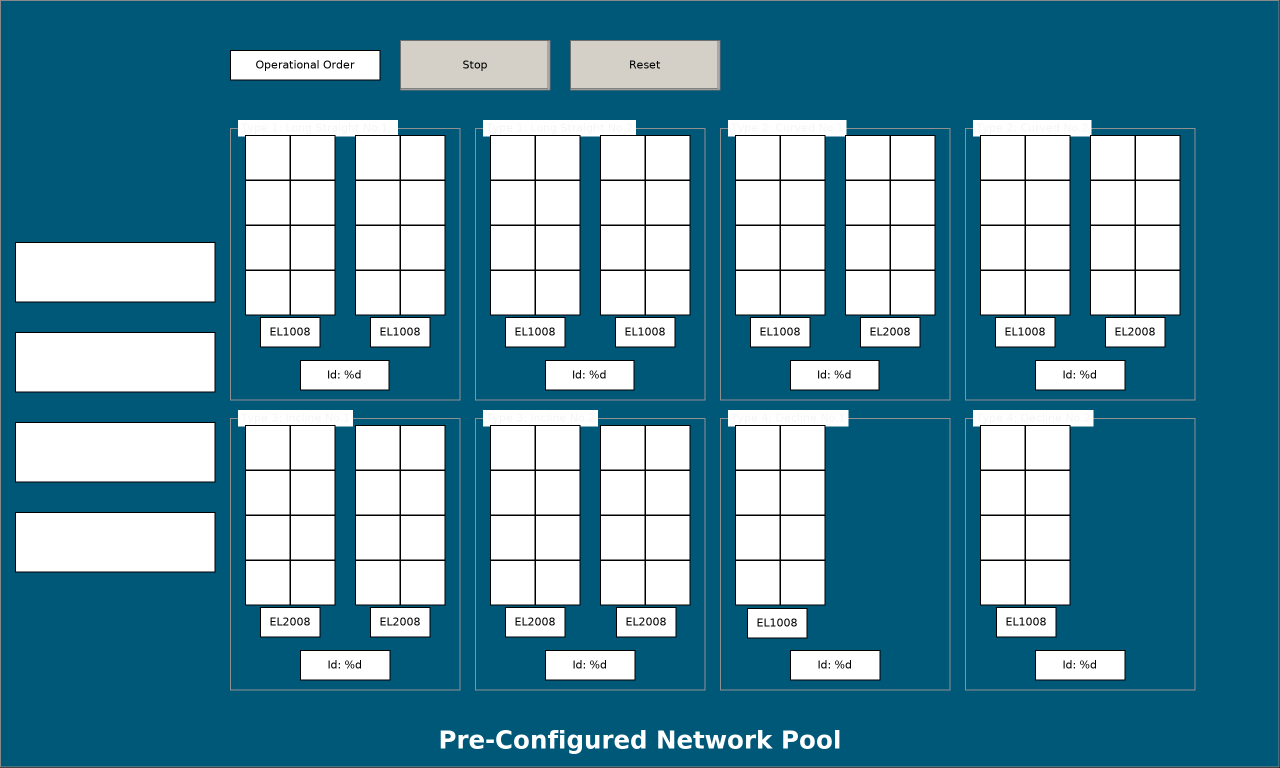
VISUALIZATION Configured  // 1280x768
    RoundedRectangle (0,0 1280x768)
    Rectangle (230,50 150x30), "Operational Order"
        OnMouseDown: change screen: Physical
    Rectangle (15,242 200x60), colour toggle: GVL_HMI.bType1Present, text list: 'RackText', text index: 11
    Rectangle (15,332 200x60), colour toggle: GVL_HMI.bType2Present, text list: 'RackText', text index: 8
    Rectangle (15,422 200x60), colour toggle: GVL_HMI.bType3Present, text list: 'RackText', text index: 9
    Rectangle (15,512 200x60), colour toggle: GVL_HMI.bType4Present, text list: 'RackText', text index: 10
    GroupBox (230,120 230x280), "Type 1: Long Straight No.1:"
        Rectangle (15,15 45x45), colour toggle: MAIN.arrFb2In[0].stRack.ST_in1.Input1
        Rectangle (15,150 45x45), colour toggle: MAIN.arrFb2In[0].stRack.ST_in1.Input7
        Rectangle (60,150 45x45), colour toggle: MAIN.arrFb2In[0].stRack.ST_in1.Input8
        Rectangle (60,15 45x45), colour toggle: MAIN.arrFb2In[0].stRack.ST_in1.Input2
        Rectangle (15,60 45x45), colour toggle: MAIN.arrFb2In[0].stRack.ST_in1.Input3
        Rectangle (60,60 45x45), colour toggle: MAIN.arrFb2In[0].stRack.ST_in1.Input4
        Rectangle (60,105 45x45), colour toggle: MAIN.arrFb2In[0].stRack.ST_in1.Input6
        Rectangle (125,15 45x45), colour toggle: MAIN.arrFb2In[0].stRack.ST_in2.Input1
        Rectangle (125,60 45x45), colour toggle: MAIN.arrFb2In[0].stRack.ST_in2.Input3
        Rectangle (125,150 45x45), colour toggle: MAIN.arrFb2In[0].stRack.ST_in2.Input7
        Rectangle (170,60 45x45), colour toggle: MAIN.arrFb2In[0].stRack.ST_in2.Input4
        Rectangle (170,150 45x45), colour toggle: MAIN.arrFb2In[0].stRack.ST_in2.Input8
        Rectangle (15,105 45x45), colour toggle: MAIN.arrFb2In[0].stRack.ST_in1.Input5
        Rectangle (30,197 60x30), "EL1008"
        Rectangle (140,197 60x30), "EL1008"
        Rectangle (170,15 45x45), colour toggle: MAIN.arrFb2In[0].stRack.ST_in2.Input2
        Rectangle (125,105 45x45), colour toggle: MAIN.arrFb2In[0].stRack.ST_in2.Input5
        Rectangle (170,105 45x45), colour toggle: MAIN.arrFb2In[0].stRack.ST_in2.Input6
        Rectangle (70,240 89x30), "Id: %d", text variable: GVL_IO.arrIds[0], colour toggle: GVL_HMI.arrPresent[0]
    GroupBox (475,120 230x280), "Type 1: Long Straight No.2"
        Rectangle (15,15 45x45), colour toggle: MAIN.arrFb2In[1].stRack.ST_in1.Input1
        Rectangle (60,15 45x45), colour toggle: MAIN.arrFb2In[1].stRack.ST_in1.Input2
        Rectangle (60,105 45x45), colour toggle: MAIN.arrFb2In[1].stRack.ST_in1.Input6
        Rectangle (60,150 45x45), colour toggle: MAIN.arrFb2In[1].stRack.ST_in1.Input8
        Rectangle (15,60 45x45), colour toggle: MAIN.arrFb2In[1].stRack.ST_in1.Input3
        Rectangle (15,105 45x45), colour toggle: MAIN.arrFb2In[1].stRack.ST_in1.Input5
        Rectangle (15,150 45x45), colour toggle: MAIN.arrFb2In[1].stRack.ST_in1.Input7
        Rectangle (60,60 45x45), colour toggle: MAIN.arrFb2In[1].stRack.ST_in1.Input4
        Rectangle (125,15 45x45), colour toggle: MAIN.arrFb2In[1].stRack.ST_in2.Input1
        Rectangle (170,15 45x45), colour toggle: MAIN.arrFb2In[1].stRack.ST_in2.Input2
        Rectangle (125,60 45x45), colour toggle: MAIN.arrFb2In[1].stRack.ST_in2.Input3
        Rectangle (170,60 45x45), colour toggle: MAIN.arrFb2In[1].stRack.ST_in2.Input4
        Rectangle (125,105 45x45), colour toggle: MAIN.arrFb2In[1].stRack.ST_in2.Input5
        Rectangle (170,105 45x45), colour toggle: MAIN.arrFb2In[1].stRack.ST_in2.Input6
        Rectangle (125,150 45x45), colour toggle: MAIN.arrFb2In[1].stRack.ST_in2.Input7
        Rectangle (170,150 45x45), colour toggle: MAIN.arrFb2In[1].stRack.ST_in2.Input8
        Rectangle (30,197 60x30), "EL1008"
        Rectangle (140,197 60x30), "EL1008"
        Rectangle (70,240 89x30), "Id: %d", text variable: GVL_IO.arrIds[1], colour toggle: GVL_HMI.arrPresent[1]
    GroupBox (720,120 230x280), "Type 2: Curved No.1"
        Rectangle (15,15 45x45), colour toggle: MAIN.arrFb1In1Out[0].stRack.ST_In.Input1
        Rectangle (60,15 45x45), colour toggle: MAIN.arrFb1In1Out[0].stRack.ST_In.Input2
        Rectangle (60,105 45x45), colour toggle: MAIN.arrFb1In1Out[0].stRack.ST_In.Input6
        Rectangle (60,150 45x45), colour toggle: MAIN.arrFb1In1Out[0].stRack.ST_In.Input8
        Rectangle (15,60 45x45), colour toggle: MAIN.arrFb1In1Out[0].stRack.ST_In.Input3
        Rectangle (15,105 45x45), colour toggle: MAIN.arrFb1In1Out[0].stRack.ST_In.Input5
        Rectangle (15,150 45x45), colour toggle: MAIN.arrFb1In1Out[0].stRack.ST_In.Input7
        Rectangle (60,60 45x45), colour toggle: MAIN.arrFb1In1Out[0].stRack.ST_In.Input4
        Rectangle (125,15 45x45), colour toggle: MAIN.arrFb1In1Out[0].stRack.ST_Out.Output1
        Rectangle (170,15 45x45), colour toggle: MAIN.arrFb1In1Out[0].stRack.ST_Out.Output2
        Rectangle (125,60 45x45), colour toggle: MAIN.arrFb1In1Out[0].stRack.ST_Out.Output3
        Rectangle (170,60 45x45), colour toggle: MAIN.arrFb1In1Out[0].stRack.ST_Out.Output4
        Rectangle (125,105 45x45), colour toggle: MAIN.arrFb1In1Out[0].stRack.ST_Out.Output5
        Rectangle (170,105 45x45), colour toggle: MAIN.arrFb1In1Out[0].stRack.ST_Out.Output6
        Rectangle (125,150 45x45), colour toggle: MAIN.arrFb1In1Out[0].stRack.ST_Out.Output7
        Rectangle (170,150 45x45), colour toggle: MAIN.arrFb1In1Out[0].stRack.ST_Out.Output8
        Rectangle (30,197 60x30), "EL1008"
        Rectangle (140,197 60x30), "EL2008"
        Rectangle (70,240 89x30), "Id: %d", text variable: GVL_IO.arrIds[2], colour toggle: GVL_HMI.arrPresent[2]
    GroupBox (965,120 230x280), "Type 2: Curved No.2"
        Rectangle (15,15 45x45), colour toggle: MAIN.arrFb1In1Out[1].stRack.ST_In.Input1
        Rectangle (60,15 45x45), colour toggle: MAIN.arrFb1In1Out[1].stRack.ST_In.Input2
        Rectangle (60,105 45x45), colour toggle: MAIN.arrFb1In1Out[1].stRack.ST_In.Input6
        Rectangle (60,150 45x45), colour toggle: MAIN.arrFb1In1Out[1].stRack.ST_In.Input8
        Rectangle (15,60 45x45), colour toggle: MAIN.arrFb1In1Out[1].stRack.ST_In.Input3
        Rectangle (15,105 45x45), colour toggle: MAIN.arrFb1In1Out[1].stRack.ST_In.Input5
        Rectangle (15,150 45x45), colour toggle: MAIN.arrFb1In1Out[1].stRack.ST_In.Input7
        Rectangle (60,60 45x45), colour toggle: MAIN.arrFb1In1Out[1].stRack.ST_In.Input4
        Rectangle (125,15 45x45), colour toggle: MAIN.arrFb1In1Out[1].stRack.ST_Out.Output1
        Rectangle (170,15 45x45), colour toggle: MAIN.arrFb1In1Out[1].stRack.ST_Out.Output2
        Rectangle (125,60 45x45), colour toggle: MAIN.arrFb1In1Out[1].stRack.ST_Out.Output3
        Rectangle (170,60 45x45), colour toggle: MAIN.arrFb1In1Out[1].stRack.ST_Out.Output4
        Rectangle (125,105 45x45), colour toggle: MAIN.arrFb1In1Out[1].stRack.ST_Out.Output5
        Rectangle (170,105 45x45), colour toggle: MAIN.arrFb1In1Out[1].stRack.ST_Out.Output6
        Rectangle (125,150 45x45), colour toggle: MAIN.arrFb1In1Out[1].stRack.ST_Out.Output7
        Rectangle (170,150 45x45), colour toggle: MAIN.arrFb1In1Out[1].stRack.ST_Out.Output8
        Rectangle (30,197 60x30), "EL1008"
        Rectangle (140,197 60x30), "EL2008"
        Rectangle (70,240 90x30), "Id: %d", text variable: GVL_IO.arrIds[3], colour toggle: GVL_HMI.arrPresent[3]
    GroupBox (720,410 230x280), "Type 4: Decline No.1"
        Rectangle (15,15 45x45), colour toggle: MAIN.arrFb1In[0].stRack.ST_In.Input1
        Rectangle (60,15 45x45), colour toggle: MAIN.arrFb1In[0].stRack.ST_In.Input2
        Rectangle (60,105 45x45), colour toggle: MAIN.arrFb1In[0].stRack.ST_In.Input6
        Rectangle (60,150 45x45), colour toggle: MAIN.arrFb1In[0].stRack.ST_In.Input8
        Rectangle (15,60 45x45), colour toggle: MAIN.arrFb1In[0].stRack.ST_In.Input3
        Rectangle (15,105 45x45), colour toggle: MAIN.arrFb1In[0].stRack.ST_In.Input5
        Rectangle (15,150 45x45), colour toggle: MAIN.arrFb1In[0].stRack.ST_In.Input7
        Rectangle (60,60 45x45), colour toggle: MAIN.arrFb1In[0].stRack.ST_In.Input4
        Rectangle (27,198 60x30), "EL1008"
        Rectangle (70,240 90x30), "Id: %d", text variable: GVL_IO.arrIds[6], colour toggle: GVL_HMI.arrPresent[6]
    GroupBox (230,410 230x280), "Type 3: Incline No.1"
        Rectangle (15,15 45x45), colour toggle: MAIN.arrFb2Out[0].stRack.ST_Out1.Output1
        Rectangle (60,15 45x45), colour toggle: MAIN.arrFb2Out[0].stRack.ST_Out1.Output2
        Rectangle (60,105 45x45), colour toggle: MAIN.arrFb2Out[0].stRack.ST_Out1.Output6
        Rectangle (60,150 45x45), colour toggle: MAIN.arrFb2Out[0].stRack.ST_Out1.Output8
        Rectangle (15,60 45x45), colour toggle: MAIN.arrFb2Out[0].stRack.ST_Out1.Output3
        Rectangle (15,105 45x45), colour toggle: MAIN.arrFb2Out[0].stRack.ST_Out1.Output5
        Rectangle (15,150 45x45), colour toggle: MAIN.arrFb2Out[0].stRack.ST_Out1.Output7
        Rectangle (60,60 45x45), colour toggle: MAIN.arrFb2Out[0].stRack.ST_Out1.Output4
        Rectangle (125,15 45x45), colour toggle: MAIN.arrFb2Out[0].stRack.ST_Out2.Output1
        Rectangle (170,15 45x45), colour toggle: MAIN.arrFb2Out[0].stRack.ST_Out2.Output2
        Rectangle (125,60 45x45), colour toggle: MAIN.arrFb2Out[0].stRack.ST_Out2.Output3
        Rectangle (170,60 45x45), colour toggle: MAIN.arrFb2Out[0].stRack.ST_Out2.Output4
        Rectangle (125,105 45x45), colour toggle: MAIN.arrFb2Out[0].stRack.ST_Out2.Output5
        Rectangle (170,105 45x45), colour toggle: MAIN.arrFb2Out[0].stRack.ST_Out2.Output6
        Rectangle (125,150 45x45), colour toggle: MAIN.arrFb2Out[0].stRack.ST_Out2.Output7
        Rectangle (170,150 45x45), colour toggle: MAIN.arrFb2Out[0].stRack.ST_Out2.Output8
        Rectangle (30,197 60x30), "EL2008"
        Rectangle (140,197 60x30), "EL2008"
        Rectangle (70,240 90x30), "Id: %d", text variable: GVL_IO.arrIds[4], colour toggle: GVL_HMI.arrPresent[4]
    GroupBox (475,410 230x280), "Type 3: Incline No.2"
        Rectangle (15,15 45x45), colour toggle: MAIN.arrFb2Out[1].stRack.ST_Out1.Output1
        Rectangle (60,15 45x45), colour toggle: MAIN.arrFb2Out[1].stRack.ST_Out1.Output2
        Rectangle (60,105 45x45), colour toggle: MAIN.arrFb2Out[1].stRack.ST_Out1.Output6
        Rectangle (60,150 45x45), colour toggle: MAIN.arrFb2Out[1].stRack.ST_Out1.Output8
        Rectangle (15,60 45x45), colour toggle: MAIN.arrFb2Out[1].stRack.ST_Out1.Output2
        Rectangle (15,105 45x45), colour toggle: MAIN.arrFb2Out[1].stRack.ST_Out1.Output5
        Rectangle (15,150 45x45), colour toggle: MAIN.arrFb2Out[1].stRack.ST_Out1.Output7
        Rectangle (60,60 45x45), colour toggle: MAIN.arrFb2Out[1].stRack.ST_Out1.Output4
        Rectangle (125,15 45x45), colour toggle: MAIN.arrFb2Out[1].stRack.ST_Out2.Output1
        Rectangle (125,60 45x45), colour toggle: MAIN.arrFb2Out[1].stRack.ST_Out2.Output3
        Rectangle (170,60 45x45), colour toggle: MAIN.arrFb2Out[1].stRack.ST_Out2.Output4
        Rectangle (125,105 45x45), colour toggle: MAIN.arrFb2Out[1].stRack.ST_Out2.Output5
        Rectangle (170,105 45x45), colour toggle: MAIN.arrFb2Out[1].stRack.ST_Out2.Output6
        Rectangle (125,150 45x45), colour toggle: MAIN.arrFb2Out[1].stRack.ST_Out2.Output7
        Rectangle (170,150 45x45), colour toggle: MAIN.arrFb2Out[1].stRack.ST_Out2.Output8
        Rectangle (30,197 60x30), "EL2008"
        Rectangle (141,197 60x30), "EL2008"
        Rectangle (170,15 45x45), colour toggle: MAIN.arrFb2Out[1].stRack.ST_Out2.Output2
        Rectangle (70,240 90x30), "Id: %d", text variable: GVL_IO.arrIds[5], colour toggle: GVL_HMI.arrPresent[5]
    GroupBox (965,410 230x280), "Type 4: Decline No.2"
        Rectangle (15,15 45x45), colour toggle: MAIN.arrFb1In[1].stRack.ST_In.Input1
        Rectangle (60,15 45x45), colour toggle: MAIN.arrFb1In[1].stRack.ST_In.Input2
        Rectangle (60,105 45x45), colour toggle: MAIN.arrFb1In[1].stRack.ST_In.Input6
        Rectangle (60,150 45x45), colour toggle: MAIN.arrFb1In[1].stRack.ST_In.Input8
        Rectangle (15,60 45x45), colour toggle: MAIN.arrFb1In[1].stRack.ST_In.Input3
        Rectangle (15,105 45x45), colour toggle: MAIN.arrFb1In[1].stRack.ST_In.Input5
        Rectangle (15,150 45x45), colour toggle: MAIN.arrFb1In[1].stRack.ST_In.Input7
        Rectangle (60,60 45x45), colour toggle: MAIN.arrFb1In[1].stRack.ST_In.Input4
        Rectangle (31,197 60x30), "EL1008"
        Rectangle (70,240 90x30), "Id: %d", text variable: GVL_IO.arrIds[7], colour toggle: GVL_HMI.arrPresent[7]
    Button (400,40 150x50), "Stop"
        tap MAIN.bStop
    Button (570,40 150x50), "Reset"
        tap MAIN.bReset
    Label (0,725 1280x30), "Pre-Configured Network Pool"
END_VISUALIZATION

(* stored: Version 1.1.0.1, ProductVersion 3.1.4024.6
   Visu Configured: Id {adec3cce-f487-454d-b5b9-d31302fe0b64} *)
